{attribute 'qualified_only'}
VAR_GLOBAL
	AlarmTexts: ARRAY [0..999] OF STRING;
END_VAR

(* stored: Version 1.1.0.1
   GVL HMI_Texts: Id {df75cf03-87bc-4abf-bcb4-a88c4ad2ee73} *)
